FUNCTION_BLOCK FaultLatch (* Basic Function Block Type *)
  (* Standard: 61499-2 *)
  (* Version 0.0, 2/24/2026, Schneider Electric, Template *)
  PACKAGE Main;
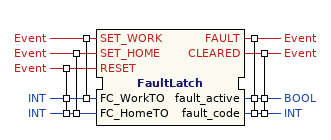
  EVENT_INPUT
    SET_WORK WITH FC_WorkTO;
    SET_HOME WITH FC_HomeTO;
    RESET WITH FC_WorkTO, FC_HomeTO;
  END_EVENT
  EVENT_OUTPUT
    FAULT WITH fault_active, fault_code; (* Fires when fault becomes active *)
    CLEARED WITH fault_active, fault_code;
  END_EVENT
  VAR_INPUT
    FC_WorkTO : INT := 1001; (* Input event qualifier *)
    FC_HomeTO : INT := 1002;
  END_VAR
  VAR_OUTPUT
    fault_active : BOOL;
    fault_code : INT;
  END_VAR
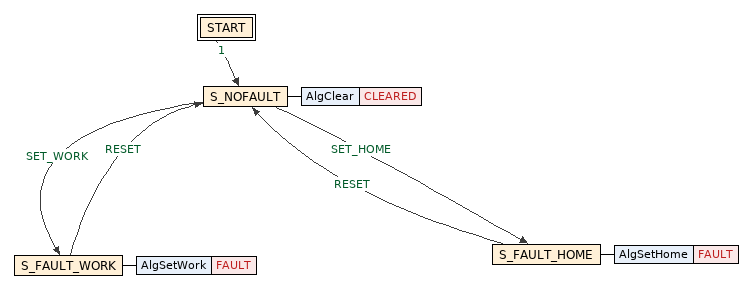
  EC_STATES
    START; (* Initial State *)
    S_NOFAULT : AlgClear -> CLEARED;
    S_FAULT_WORK : AlgSetWork -> FAULT;
    S_FAULT_HOME : AlgSetHome -> FAULT;
  END_STATES
  EC_TRANSITIONS
    START TO S_NOFAULT := 1;
    S_NOFAULT TO S_FAULT_WORK := SET_WORK;
    S_NOFAULT TO S_FAULT_HOME := SET_HOME;
    S_FAULT_WORK TO S_NOFAULT := RESET;
    S_FAULT_HOME TO S_NOFAULT := RESET;
  END_TRANSITIONS
  ALGORITHM AlgClear IN ST:
fault_active := FALSE;
fault_code := 0;
  END_ALGORITHM
  ALGORITHM AlgSetWork IN ST:
fault_active := TRUE;
fault_code := FC_WorkTO;
  END_ALGORITHM
  ALGORITHM AlgSetHome IN ST:
fault_active := TRUE;
fault_code := FC_HomeTO;
  END_ALGORITHM
END_FUNCTION_BLOCK
